(* IEC 61131-3 sources: plc-vscode/tests/st/test-ready/trust-platform/examples/plcopen_xml_st_complete/src, 3 files *)

(* ---- types.st ---- *)
TYPE
  PumpMode : (Stopped := 0, Running := 1, Fault := 2);
  PumpConfig : STRUCT
    RampTime : TIME := T#2s;
    MaxStartsPerHour : UINT := 10;
  END_STRUCT;
  PumpIndex : INT(1..16);
  PumpAlarmLatch : ARRAY[1..4] OF BOOL;
END_TYPE

(* ---- main.st ---- *)
PROGRAM Main
VAR
    Controller : PumpController;
    StartCmd : BOOL := TRUE;
END_VAR

Controller(Enable := StartCmd);
END_PROGRAM

FUNCTION_BLOCK PumpController
VAR_INPUT
    Enable : BOOL;
END_VAR
VAR
    Config : PumpConfig;
    RunTimer : TON;
END_VAR

RunTimer(IN := Enable, PT := Config.RampTime);
END_FUNCTION_BLOCK

(* ---- configuration.st ---- *)
CONFIGURATION PlantConfig
RESOURCE Cpu0 ON CPU
    TASK FastTask (INTERVAL := T#100ms, PRIORITY := 1);
    PROGRAM Main WITH FastTask : Main;
END_RESOURCE
END_CONFIGURATION
